PROGRAM MAIN
VAR
	
	B_out :BOOL;
	B_in  :BOOL;

END_VAR

P0_Start_Initialization();
B_out := B_in;

END_PROGRAM

(* stored: Version 1.1.0.1, ProductVersion 3.1.4022.7
   POU MAIN: Id {bdcc1b68-15b5-4f79-971c-4d1d2ef04cb5}, SpecialFunc None *)
